FUNCTION_BLOCK Mixer_Timer (* Composite FB wrapping other FBs *)
  (* Standard: 61499-2 *)
  (* Version 1.0, 2024-02-16, ADMIN *)
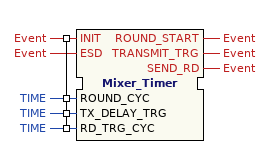
  EVENT_INPUT
    INIT WITH ROUND_CYC, TX_DELAY_TRG, RD_TRG_CYC; (* Initialization Request *)
    ESD; (* Normal Execution Request *)
  END_EVENT
  EVENT_OUTPUT
    ROUND_START; (* Execution Confirmation *)
    TRANSMIT_TRG;
    SEND_RD;
  END_EVENT
  VAR_INPUT
    ROUND_CYC : TIME; (* Input event qualifier *)
    TX_DELAY_TRG : TIME;
    RD_TRG_CYC : TIME;
  END_VAR
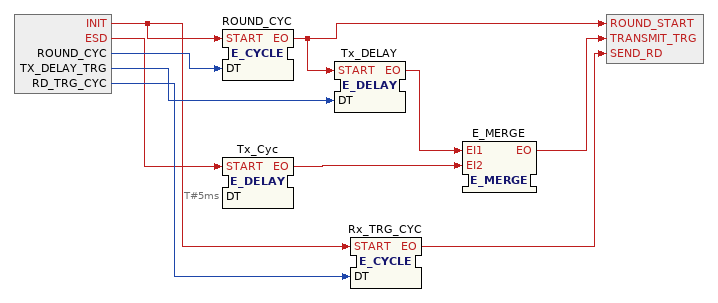
  FBS
    ROUND_CYC : E_CYCLE;
    Tx_DELAY : E_DELAY;
    E_MERGE : E_MERGE;
    Tx_Cyc : E_DELAY(DT := T#5ms);
    Rx_TRG_CYC : E_CYCLE;
  END_FBS
  EVENT_CONNECTIONS
    Tx_DELAY.EO TO E_MERGE.EI1;
    ROUND_CYC.EO TO Tx_DELAY.START;
    Tx_Cyc.EO TO E_MERGE.EI2;
    INIT TO ROUND_CYC.START;
    ROUND_CYC.EO TO ROUND_START;
    E_MERGE.EO TO TRANSMIT_TRG;
    Rx_TRG_CYC.EO TO SEND_RD;
    ESD TO Tx_Cyc.START;
    INIT TO Rx_TRG_CYC.START;
  END_CONNECTIONS
  DATA_CONNECTIONS
    ROUND_CYC TO ROUND_CYC.DT;
    TX_DELAY_TRG TO Tx_DELAY.DT;
    RD_TRG_CYC TO Rx_TRG_CYC.DT;
  END_CONNECTIONS
END_FUNCTION_BLOCK
